// TIA Portal V21 export
DATA_BLOCK "Button"   // DB2
{ S7_Optimized_Access := 'TRUE' }
// stored: MemoryReserve 100
   VAR
      start : Bool;
      stop : Bool;
      reset : Bool;
      emergencyStop : Bool;
      suspendResume : Bool;
      manualMode : Bool;
      manualRed : Bool;
      manualYellow : Bool;
      manualGreen : Bool;
      Input : "ST_Button";
   END_VAR
BEGIN
END_DATA_BLOCK
